(* Schneider Machine Expert - Basic project animation moving, file version 2.7.0.0 *)
(* ProjectInformations: Name=New project *)

HARDWARE
  Cpu 0: TM221CE24T
  EthernetConfiguration: NetworkName=M221, IpAllocationMode=FixedAddress, IpAddress=0.0.0.0, SubnetMask=0.0.0.0
  SerialLineConfiguration: Baud=Baud19200, Parity=ParityEven, DataBits=DataBits8, StopBits=StopBits1, PhysicalMedium=PhysicalMediumRs485, TransmissionMode=TransmissionModeModbusRtu, SlaveId=1, Addressing=SlaveAddressing
  MastTask: UsePeriodScanMode=false, PeriodScan=100
  FastTask: Period=255
  CpuBehavior: StartingMode=StartAsPreviousState, AutoSaveRamOnEeprom=true, WatchdogPeriod=250

SYMBOLS  (address, symbol, comment, settings)
  %M0       PB_ON
  %M1       PB_OFF
  %M2       MOVE_FORWARD
  %M3       MOVE_BACKWARD
  %M10      SYSTEM
  %M11      FORWARD_STATE
  %M12      BACKWARD_STATE
  %TM0        [Preset=10, Base=OneSecond]
  %TM1        [Preset=10, Base=OneSecond]

POU New POU
  (* SectionNumber=1 *)

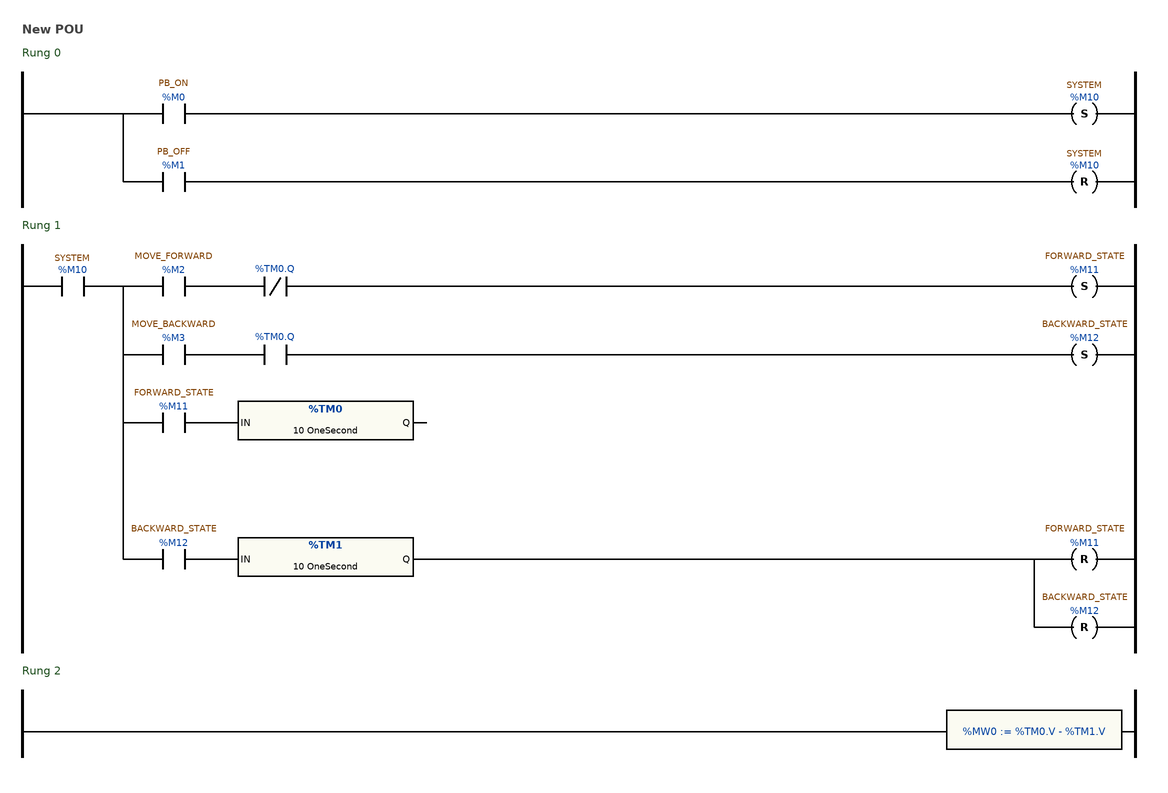

// Rung 0
  LD 1
  MPS
  AND %M0                 (* PB_ON *)
  S %M10                  (* SYSTEM *)
  MPP
  AND %M1                 (* PB_OFF *)
  R %M10                  (* SYSTEM *)
  // as ST:
  //   IF PB_ON THEN SYSTEM := TRUE; END_IF;
  //   IF PB_OFF THEN SYSTEM := FALSE; END_IF;

// Rung 1
  LD 1
  MULTIFB
  LD 1
  AND %M10                (* SYSTEM *)
  ST %MW2009:X0
  LD %MW2009:X0
  MPS
  AND %M2                 (* MOVE_FORWARD *)
  ANDN %TM0.Q
  S %M11                  (* FORWARD_STATE *)
  MPP
  AND %M3                 (* MOVE_BACKWARD *)
  AND %TM0.Q
  S %M12                  (* BACKWARD_STATE *)
  BLK %TM0
  LD %MW2009:X0
  AND %M11                (* FORWARD_STATE *)
  IN
  END_BLK
  BLK %TM1
  LD %MW2009:X0
  AND %M12                (* BACKWARD_STATE *)
  IN
  OUT_BLK
  LD Q
  R %M11                  (* FORWARD_STATE *)
  R %M12                  (* BACKWARD_STATE *)
  END_BLK
  MULTIFB
  // as ST:
  //   IF SYSTEM AND MOVE_FORWARD AND NOT %TM0.Q THEN FORWARD_STATE := TRUE; END_IF;
  //   IF SYSTEM AND MOVE_BACKWARD AND %TM0.Q THEN BACKWARD_STATE := TRUE; END_IF;
  //   %TM0(IN := SYSTEM AND FORWARD_STATE);
  //   %TM1(IN := SYSTEM AND BACKWARD_STATE);
  //   IF %TM1.Q THEN FORWARD_STATE := FALSE; END_IF;
  //   IF %TM1.Q THEN BACKWARD_STATE := FALSE; END_IF;

// Rung 2
  LD 1
  [ %MW0 := %TM0.V - %TM1.V ]
  // as ST:
  //   %MW0 := %TM0.V - %TM1.V;
